// TIA Portal V19 export
ORGANIZATION_BLOCK "Main"   // OB2301, LAD, ProgramCycle
TITLE = "Main Program Sweep (Cycle)"
// stored: AutoNumber false, Namespace Unit2.EM2, SetENOAutomatically false
   VAR_INPUT
      Initial_Call : Bool;   // Initial call of this OB
      Remanence : Bool;   // =True, if remanent data are available
   END_VAR
BEGIN

REGION Network 2 (SCL)
   "Unit2.EM2.instSimulation"();

   "Unit2.EM2.CallEquipment_DB"(unitStatus:="Unit2.EmNodes".unitStatus,
                    unitAlarmDB:="Unit2.Alarms".emAlarms[Unit2_EM2],
                    emFeedback:="Unit2.EmNodes".emFeedback[Unit2_EM2]);
END_REGION
END_ORGANIZATION_BLOCK
